// SIMATIC S7-200 project (STEP 7-Micro/WIN), CPU 224 REL 02.01

SYMBOL_TABLE USER1
D1               I0.2
D2               I0.1
D3               I0.3
GREEN            Q0.0
RED              Q0.1
CONVAYER         Q0.2
ACTUATOR         Q0.3
END_SYMBOL_TABLE

ORGANIZATION_BLOCK MAIN:OB1
TITLE=PROGRAM COMMENTS
BEGIN
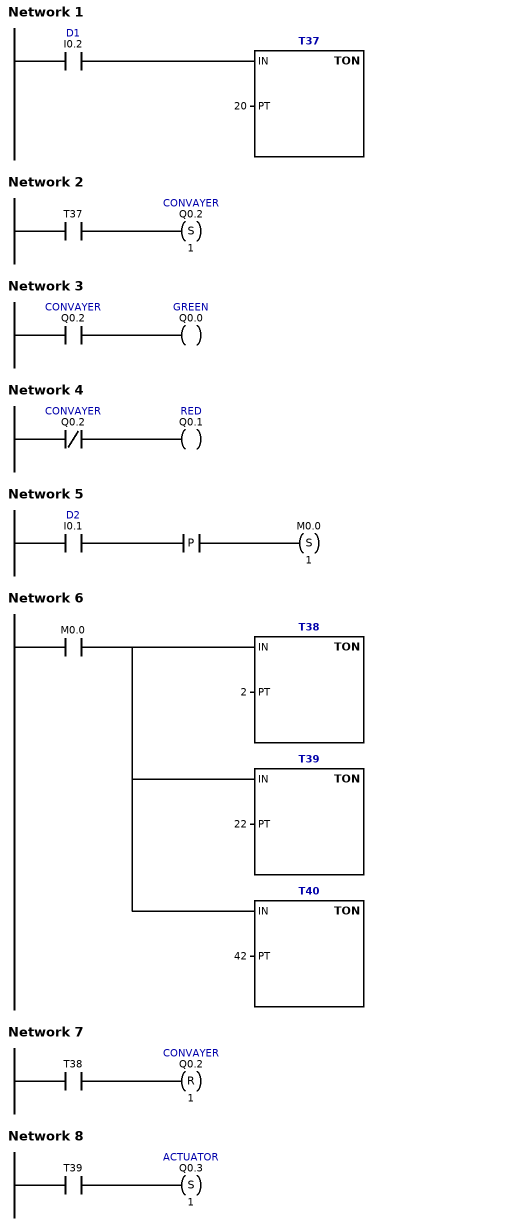
Network 1
// (network saved uncompiled; LAD cells follow)
// row 0: c0 -| |- D1:I0.2  c1 --  c2 [TON T37 IN:=power@row0, PT:=20]
// row 1: c2 [box]
Network 2
LD     T37
S      CONVAYER:Q0.2, 1
Network 3
LD     CONVAYER:Q0.2
=      GREEN:Q0.0
Network 4
LDN    CONVAYER:Q0.2
=      RED:Q0.1
Network 5
LD     D2:I0.1
EU
S      M0.0, 1
Network 6
LD     M0.0
TON    T38, 2
TON    T39, 22
TON    T40, 42
Network 7
LD     T38
R      CONVAYER:Q0.2, 1
Network 8
LD     T39
S      ACTUATOR:Q0.3, 1
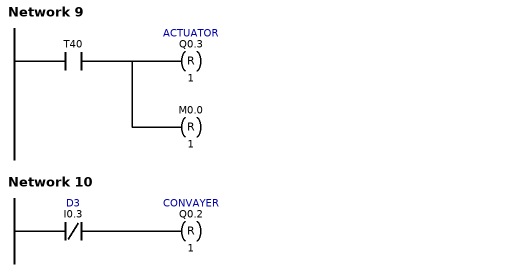
Network 9
LD     T40
R      ACTUATOR:Q0.3, 1
R      M0.0, 1
Network 10
// (network saved uncompiled; LAD cells follow)
// row 0: c0 -|/|- D3:I0.3  c1 -(R) CONVAYER:Q0.2, 1
END_ORGANIZATION_BLOCK
